FUNCTION_BLOCK  FB_FastOpen
VAR_INPUT
    MotorCenterPosition : INT;           // P0 (open pos)
    C2 : INT;                            // Encoder actual count
END_VAR
VAR_IN_OUT
    EncoderShadow : INT;                 // Cs (shadow register)
    SlitStatusFlag : INT;                // Df
END_VAR
VAR_OUTPUT
    Complete : BOOL := FALSE;
END_VAR
VAR
    State : INT := 0; // 0: idle, 1: moving, 2: done
END_VAR

METHOD Execute : BOOL
VAR_INPUT
END_VAR
IF State = 0 THEN
    // Start movement to open (simulate instant success; call MC_MoveAbsolute in real system)
    State := 1;
    Complete := FALSE;
ELSIF State = 1 THEN
    // Simulate motion complete; check actual motion in real system
    EncoderShadow := C2;
    SlitStatusFlag := 0;      // Open
    State := 2;
    Complete := TRUE;
END_IF
END_METHOD

METHOD Reset : BOOL
VAR_INPUT
END_VAR
    State := 0;
    Complete := FALSE;
END_METHOD

END_FUNCTION_BLOCK

(* stored: Version 1.1.0.1
   POU FB_FastOpen: Id {c73d2697-7522-4d8d-b835-3670f2667cbf}, SpecialFunc None
   Method Execute: Id {eb783105-8088-47a1-b1bf-6fcac722cbcb}
   Method Reset: Id {0da11e5b-aeee-4483-a1a2-5989efc86cfd} *)
